Yaskawa INFORM job: GO-PARK.JBI

/JOB
//NAME GO-PARK
///FOLDERNAME FOLDER001
//POS
///NPOS 0,0,0,1,0,0
///TOOL 1
///POSTYPE ROBOT
///RECTAN
///RCONF 0,0,0,0,0,0,0,0,0,0,0,0,0,0,0,0,0,0,0,0,0,0,0,0
P00091=95.757,118.537,704.751,11.1321,-47.2188,101.9621
//INST
///DATE 2025/09/30 16:22
///ATTR SC,RW
///GROUP1 RB1
NOP
MOVJ P091 VJ=100.00 PL=3
END
